Staubli VAL3: trajectory.pjx

--- trajectory.pjx ---
Parameters version=s7.2.1 stackSize=5000 millimeterUnit=true
Data file=trajectory.dtx
Library alias=io path=Disk://io/io.pjx

--- trajectory.dtx ---
public num distance
public num moveType
public num nFrameIndex = 1
public num nGasPressure
public num nIndexGun
public num nLaserPower
public num nStop
public num nTcpAction
public num nTime
public num nPWMPercent
public num nJointMode
public string comment
public string instruction
public bool toStop
public frame fTrack = {x=23, z=-50, fatherId=world[0]}
public mdesc nom_speed = {accel=200, vel=200, decel=200, tmax=300, rmax=9999, leave=30, reach=30}
